FUNCTION TryConvert_WORD_TO_LREAL : BOOL
VAR_INPUT
	in : WORD;
	out : REFERENCE TO LREAL;
END_VAR

out := WORD_TO_LREAL(in);
TryConvert_WORD_TO_LREAL := TRUE;

END_FUNCTION

(* stored: Version 1.1.0.1, ProductVersion 3.1.4024.12
   POU TryConvert_WORD_TO_LREAL: Id {0364d126-715e-4574-a3b1-6b45fd95a2c1}, SpecialFunc None *)
